FUNCTION_BLOCK PutText (* openCV text drawer *)
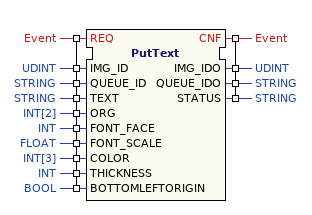
  EVENT_INPUT
    REQ WITH IMG_ID, QUEUE_ID, TEXT, ORG, FONT_FACE, FONT_SCALE, COLOR, THICKNESS, BOTTOMLEFTORIGIN;
  END_EVENT
  EVENT_OUTPUT
    CNF WITH IMG_IDO, QUEUE_IDO, STATUS;
  END_EVENT
  VAR_INPUT
    IMG_ID : UDINT;
    QUEUE_ID : STRING;
    TEXT : STRING;
    ORG : ARRAY [0..1] OF INT;
    FONT_FACE : INT;
    FONT_SCALE : FLOAT;
    COLOR : ARRAY [0..2] OF INT;
    THICKNESS : INT;
    BOTTOMLEFTORIGIN : BOOL;
  END_VAR
  VAR_OUTPUT
    IMG_IDO : UDINT;
    QUEUE_IDO : STRING;
    STATUS : STRING;
  END_VAR
END_FUNCTION_BLOCK
